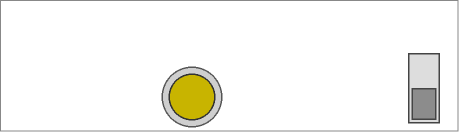
VISUALIZATION Visualization  // 459x132
    Lamp1 (157,62 70x70), variable: GVL.lamp, style: Lamp-Lamp1-Yellow
    DipSwitch (389,53 70x70), variable: GVL.knop, behaviour: TOGGLE, style: Switch-DipSwitch-Gray
END_VISUALIZATION

(* stored: Version 1.1.0.1, ProductVersion 3.1.4024.12
   Visu Visualization: Id {d862a015-9ccc-4401-92c1-f9de8a886e24} *)
